// TIA Portal V19 export
FUNCTION_BLOCK "Area"   // FB100, LAD
TITLE = AREA MANAGER / ZONE CYCLE
// v1.1 : Normal Stop required added in AreaInterface
// stored: Access Published, MemoryReserve 100, SetENOAutomatically false
   VAR_INPUT
      Estop : Bool;   // Emergency stop pressed (0=OK)
      DataIn : Struct
         SelMan : Bool;   // IN: Mode selectot in AUTO position / Select Manual mode
         SelAut : Bool;   // in quale tabella di lavoro è stato copiato / Select Auto mode
         PbStart : Bool;   // IN: Push button ACKNOWLEDGE/RESET ALARMS / Pb Start Cycle
         PbStop : Bool;   // IN: Push button START CYLE / Pb Stop Cycle
         PbStopProgrammed : Bool;   // Normally not used
         PbAckRst : Bool;   // IN: Mode selectot in MANU position / Pb Reset alarms
      END_STRUCT;
      Config : "AreaConfig";
      MachinesStatus : "MachineStatus";
      ForceStopInPhase : Bool;   // Force area in stop in phase (From PLC command)
      ForceStopProgrammed : Bool;   // Force area in stop programmed (From PLC command)
      ResetTimersTimeoutStops : Bool;   // Reset timeout of stop in phase and stop programmed
   END_VAR
   VAR_OUTPUT
      AreaInterface { ExternalVisible := 'False'; ExternalWritable := 'False'} : "AreaInterface";
      DataOut : Struct
         horn : Bool;   // Area tower acustic signal
         lampReady : Bool;   // Ready for cycle lamp
         lampCycle : Bool;   // Cylce on lamp
         LampWarningPresence : Bool;   // Area tower wanring lamp
         LampAlarmPresence : Bool;   // Area tower alarm lamp
      END_STRUCT;
      SilencingAlarms : Bool;   // Command to message manager for silecing alarms
      HMI_StatusDinamicText : Int;   // Status of area for HMI
   END_VAR
   VAR
      pbStartOneShotAux : Bool;
      RstAlrOneShot1 : Bool;
      RstAlrOneShot2 : Bool;
      CycleStopImmediately : Bool;
      CycleStopInPhase : Bool;
      CycleStarted : Bool;
      CycleStopProgrammed : Bool;
      CycleOn : Bool;
      ManAuxPe : Bool;
      ManAuxNe : Bool;
      ManPositiveEdge : Bool;
      ManNegativeEdge : Bool;
      AutAuxPe : Bool;
      AutAuxNe : Bool;
      AutPositiveEdge : Bool;
      AutNegativeEdge : Bool;
      AlarmLAuxPe : Bool;
      CycleAuxPe : Bool;
      ResetAlarmsCmd : Bool;
      tonDelayPbStart { S7_SetPoint := 'True'} : IEC_TIMER;
      tonDelayRstAck { S7_SetPoint := 'True'} : IEC_TIMER;
      tonTimeOutStopPhase { S7_SetPoint := 'True'} : IEC_TIMER;
      tonTimeOutStopProgr { S7_SetPoint := 'True'} : IEC_TIMER;
      tonTimeOutResetAlr { S7_SetPoint := 'True'} : IEC_TIMER;
   END_VAR
   VAR_TEMP
      AreaEStop : Bool;
      ManMode : Bool;
      AutMode : Bool;
      pbStartOneShot : Bool;
      CycleStop : Bool;
      CycleCheckStartCnd : Bool;
      PbAckRstDelayed : Bool;
      TimeOutPT : Time;
   END_VAR
   VAR CONSTANT
      HMI_STATUS_CODE_00_INVALID : Int := 0;
      HMI_STATUS_CODE_01_EMERGENCY : Int := 1;
      HMI_STATUS_CODE_02_SEL_0 : Int := 2;
      HMI_STATUS_CODE_11_MAN : Int := 11;
      HMI_STATUS_CODE_21_AUT_NOT_READY : Int := 21;
      HMI_STATUS_CODE_22_AUT_READY : Int := 22;
      HMI_STATUS_CODE_31_CYCLE_STARTING : Int := 31;
      HMI_STATUS_CODE_32_CYCLE_ON : Int := 32;
      HMI_STATUS_CODE_41_STOP_IMMEDIATELY : Int := 41;
      HMI_STATUS_CODE_42_STOP_IN_PHASE : Int := 42;
      HMI_STATUS_CODE_43_STOP_PROGRAMMED : Int := 43;
   END_VAR
   VAR_TEMP   // added for the SCL form of the ladder/FBD networks
      _w1 : Bool;
      _w2 : Bool;
   END_VAR
BEGIN

REGION Network 1 (SCL): Info
   //=============================================================================
   //PM FORMING
   //-----------------------------------------------------------------------------
   // Library: StandardBlocks
   // Tested with: S7-1518TF
   // Engineering: TIA Portal V18
   // Restrictions: -
   // Requirements: S7-1500
   // Functionality: Area Manager
   //
   // v1.0.0  28/12/2022 
   //=============================================================================
END_REGION

REGION Network 3: EStop active
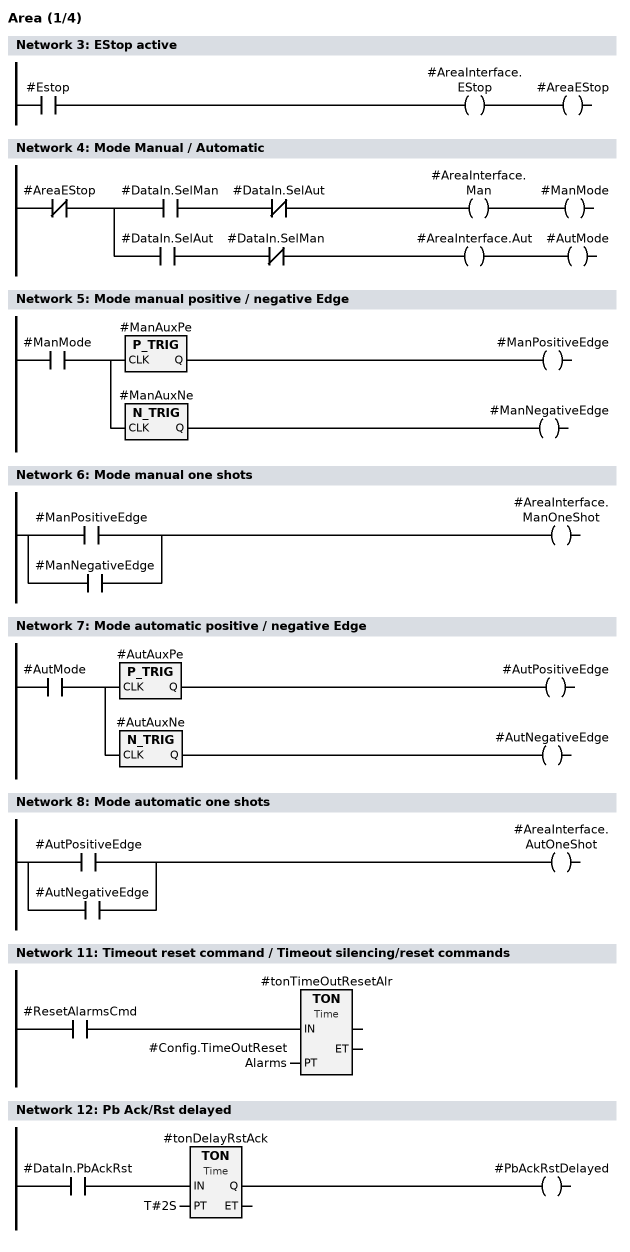
   RUNG wire#powerrail
      Contact( #Estop )
      Coil( #AreaInterface.EStop )
      Coil( #AreaEStop )
   END_RUNG
   // the same network as SCL:
   #AreaInterface.EStop := #Estop;
   #AreaEStop := #Estop;
END_REGION

REGION Network 4: Mode Manual / Automatic
   RUNG wire#powerrail
      I_Contact( #AreaEStop )
      wire#w1
      Contact( #DataIn.SelMan )
      I_Contact( #DataIn.SelAut )
      Coil( #AreaInterface.Man )
      Coil( #ManMode )
   END_RUNG
   RUNG wire#w1
      Contact( #DataIn.SelAut )
      I_Contact( #DataIn.SelMan )
      Coil( #AreaInterface.Aut )
      Coil( #AutMode )
   END_RUNG
   // the same network as SCL:
   #AreaInterface.Man := NOT #AreaEStop AND #DataIn.SelMan AND NOT #DataIn.SelAut;
   #ManMode := #AreaInterface.Man;
   #AreaInterface.Aut := NOT #AreaEStop AND #DataIn.SelAut AND NOT #DataIn.SelMan;
   #AutMode := #AreaInterface.Aut;
END_REGION

REGION Network 5: Mode manual positive / negative Edge
   RUNG wire#powerrail
      Contact( #ManMode )
      wire#w1
      P_Trig( #ManAuxPe )
      Coil( #ManPositiveEdge )
   END_RUNG
   RUNG wire#w1
      N_Trig( #ManAuxNe )
      Coil( #ManNegativeEdge )
   END_RUNG
   // the same network as SCL:
   #_w1 := #ManMode AND NOT #ManAuxPe;   // rising edge
   #ManAuxPe := #ManMode;
   #ManPositiveEdge := #_w1;
   #_w2 := NOT #ManMode AND #ManAuxNe;   // falling edge
   #ManAuxNe := #ManMode;
   #ManNegativeEdge := #_w2;
END_REGION

REGION Network 6: Mode manual one shots
   RUNG wire#powerrail
      Contact( #ManPositiveEdge )
      wire#w1
      Coil( #AreaInterface.ManOneShot )
   END_RUNG
   RUNG wire#powerrail
      Contact( #ManNegativeEdge )
   END_RUNG wire#w1
   // the same network as SCL:
   #AreaInterface.ManOneShot := #ManPositiveEdge OR #ManNegativeEdge;
END_REGION

REGION Network 7: Mode automatic positive / negative Edge
   RUNG wire#powerrail
      Contact( #AutMode )
      wire#w1
      P_Trig( #AutAuxPe )
      Coil( #AutPositiveEdge )
   END_RUNG
   RUNG wire#w1
      N_Trig( #AutAuxNe )
      Coil( #AutNegativeEdge )
   END_RUNG
   // the same network as SCL:
   #_w1 := #AutMode AND NOT #AutAuxPe;   // rising edge
   #AutAuxPe := #AutMode;
   #AutPositiveEdge := #_w1;
   #_w2 := NOT #AutMode AND #AutAuxNe;   // falling edge
   #AutAuxNe := #AutMode;
   #AutNegativeEdge := #_w2;
END_REGION

REGION Network 8: Mode automatic one shots
   RUNG wire#powerrail
      Contact( #AutPositiveEdge )
      wire#w1
      Coil( #AreaInterface.AutOneShot )
   END_RUNG
   RUNG wire#powerrail
      Contact( #AutNegativeEdge )
   END_RUNG wire#w1
   // the same network as SCL:
   #AreaInterface.AutOneShot := #AutPositiveEdge OR #AutNegativeEdge;
END_REGION

REGION Network 10: <<< ALARMS SILENCING & RESETTING >>>
END_REGION

REGION Network 11: Timeout reset command / Timeout silencing/reset commands
   RUNG wire#powerrail
      Contact( #ResetAlarmsCmd )
      { S7_Templates := "time_type := Time" } #tonTimeOutResetAlr.TON(pt := #Config.TimeOutResetAlarms, et =>)
   END_RUNG
   // the same network as SCL:
   #tonTimeOutResetAlr.TON(IN := #ResetAlarmsCmd, PT := #Config.TimeOutResetAlarms);
END_REGION

REGION Network 12: Pb Ack/Rst delayed
   RUNG wire#powerrail
      Contact( #DataIn.PbAckRst )
      { S7_Templates := "time_type := Time" } #tonDelayRstAck.TON(pt := T#2S, et =>)
      Coil( #PbAckRstDelayed )
   END_RUNG
   // the same network as SCL:
   #tonDelayRstAck.TON(IN := #DataIn.PbAckRst, PT := T#2S);
   #PbAckRstDelayed := #tonDelayRstAck.Q;
END_REGION

REGION Network 13: Alarms reset command (need ACK)
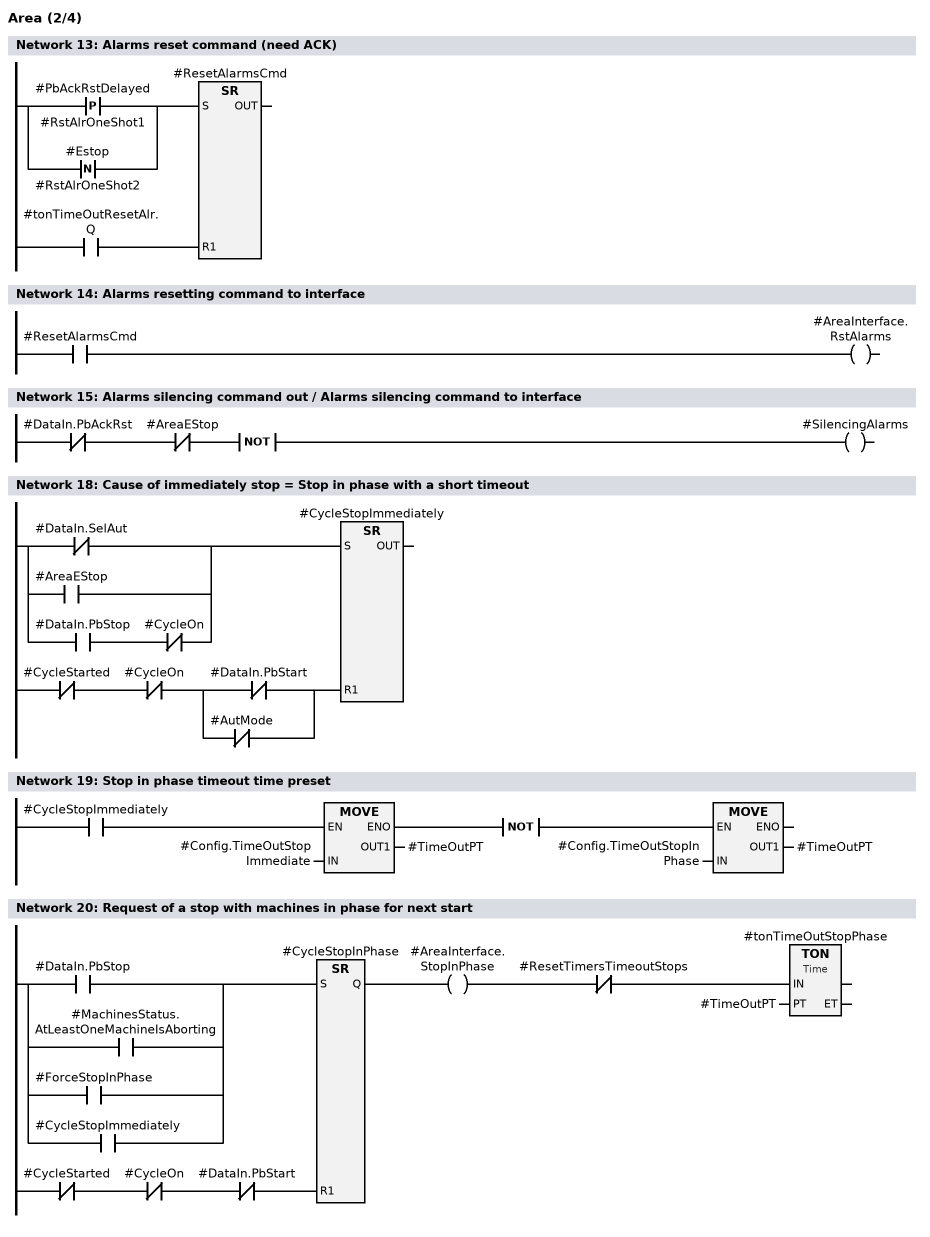
   RUNG wire#powerrail
      P_Contact(operand := #PbAckRstDelayed, bit := #RstAlrOneShot1)
      wire#w1
      S_SR(operand := #ResetAlarmsCmd, r1 := wire#w2)
   END_RUNG
   RUNG wire#powerrail
      N_Contact(operand := #Estop, bit := #RstAlrOneShot2)
   END_RUNG wire#w1
   RUNG wire#powerrail
      Contact( #tonTimeOutResetAlr.Q )
   END_RUNG wire#w2
   // the same network as SCL:
   #_w1 := #PbAckRstDelayed AND NOT #RstAlrOneShot1;   // rising edge of #PbAckRstDelayed
   #RstAlrOneShot1 := #PbAckRstDelayed;
   #_w2 := NOT #Estop AND #RstAlrOneShot2;   // falling edge of #Estop
   #RstAlrOneShot2 := #Estop;
   IF #_w1 OR #_w2 THEN
       #ResetAlarmsCmd := TRUE;   // SR flip-flop
   END_IF;
   IF #tonTimeOutResetAlr.Q THEN #ResetAlarmsCmd := FALSE; END_IF;
END_REGION

REGION Network 14: Alarms resetting command to interface
   RUNG wire#powerrail
      Contact( #ResetAlarmsCmd )
      Coil( #AreaInterface.RstAlarms )
   END_RUNG
   // the same network as SCL:
   #AreaInterface.RstAlarms := #ResetAlarmsCmd;
END_REGION

REGION Network 15: Alarms silencing command out / Alarms silencing command to interface
   RUNG wire#powerrail
      I_Contact( #DataIn.PbAckRst )
      I_Contact( #AreaEStop )
      Not()
      Coil( #SilencingAlarms )
   END_RUNG
   // the same network as SCL:
   #SilencingAlarms := NOT (NOT #DataIn.PbAckRst AND NOT #AreaEStop);
END_REGION

REGION Network 17: <<< AUTOMATIC CYCLE >>>
END_REGION

REGION Network 18: Cause of immediately stop = Stop in phase with a short timeout
   RUNG wire#powerrail
      I_Contact( #DataIn.SelAut )
      wire#w1
      S_SR(operand := #CycleStopImmediately, r1 := wire#w3)
   END_RUNG
   RUNG wire#powerrail
      Contact( #AreaEStop )
   END_RUNG wire#w1
   RUNG wire#powerrail
      Contact( #DataIn.PbStop )
      I_Contact( #CycleOn )
   END_RUNG wire#w1
   RUNG wire#powerrail
      I_Contact( #CycleStarted )
      I_Contact( #CycleOn )
      wire#w2
      I_Contact( #DataIn.PbStart )
   END_RUNG wire#w3
   RUNG wire#w2
      I_Contact( #AutMode )
   END_RUNG wire#w3
   // the same network as SCL:
   IF NOT #DataIn.SelAut OR #AreaEStop OR (#DataIn.PbStop AND NOT #CycleOn) THEN
       #CycleStopImmediately := TRUE;   // SR flip-flop
   END_IF;
   IF NOT #CycleStarted AND NOT #CycleOn AND (NOT #DataIn.PbStart OR NOT #AutMode) THEN
       #CycleStopImmediately := FALSE;
   END_IF;
END_REGION

REGION Network 19: Stop in phase timeout time preset
   RUNG wire#powerrail
      Contact( #CycleStopImmediately )
      { S7_GenerateENO := "TRUE" } Move(in := #Config.TimeOutStopImmediate, out1 => #TimeOutPT)
      Not()
      { S7_GenerateENO := "TRUE" } Move(in := #Config.TimeOutStopInPhase, out1 => #TimeOutPT)
   END_RUNG
   // the same network as SCL:
   // ENO of a box is taken as its EN; it also drops when the box reports an error
   IF #CycleStopImmediately THEN #TimeOutPT := #Config.TimeOutStopImmediate; END_IF;
   IF NOT #CycleStopImmediately THEN #TimeOutPT := #Config.TimeOutStopInPhase; END_IF;
END_REGION

REGION Network 20: Request of a stop with machines in phase for next start
   RUNG wire#powerrail
      Contact( #DataIn.PbStop )
      wire#w1
      S_SR(operand := #CycleStopInPhase, r1 := wire#w2)
      Coil( #AreaInterface.StopInPhase )
      I_Contact( #ResetTimersTimeoutStops )
      { S7_Templates := "time_type := Time" } #tonTimeOutStopPhase.TON(pt := #TimeOutPT, et =>)
   END_RUNG
   RUNG wire#powerrail
      Contact( #MachinesStatus.AtLeastOneMachineIsAborting )
   END_RUNG wire#w1
   RUNG wire#powerrail
      Contact( #ForceStopInPhase )
   END_RUNG wire#w1
   RUNG wire#powerrail
      Contact( #CycleStopImmediately )
   END_RUNG wire#w1
   RUNG wire#powerrail
      I_Contact( #CycleStarted )
      I_Contact( #CycleOn )
      I_Contact( #DataIn.PbStart )
   END_RUNG wire#w2
   // the same network as SCL:
   IF #DataIn.PbStop OR #MachinesStatus.AtLeastOneMachineIsAborting OR #ForceStopInPhase OR #CycleStopImmediately THEN
       #CycleStopInPhase := TRUE;   // SR flip-flop
   END_IF;
   IF NOT #CycleStarted AND NOT #CycleOn AND NOT #DataIn.PbStart THEN #CycleStopInPhase := FALSE; END_IF;
   #AreaInterface.StopInPhase := #CycleStopInPhase;
   #tonTimeOutStopPhase.TON(IN := #CycleStopInPhase AND NOT #ResetTimersTimeoutStops, PT := #TimeOutPT);
END_REGION

REGION Network 21: Request of a programmed stop (e.g. at the end of part)
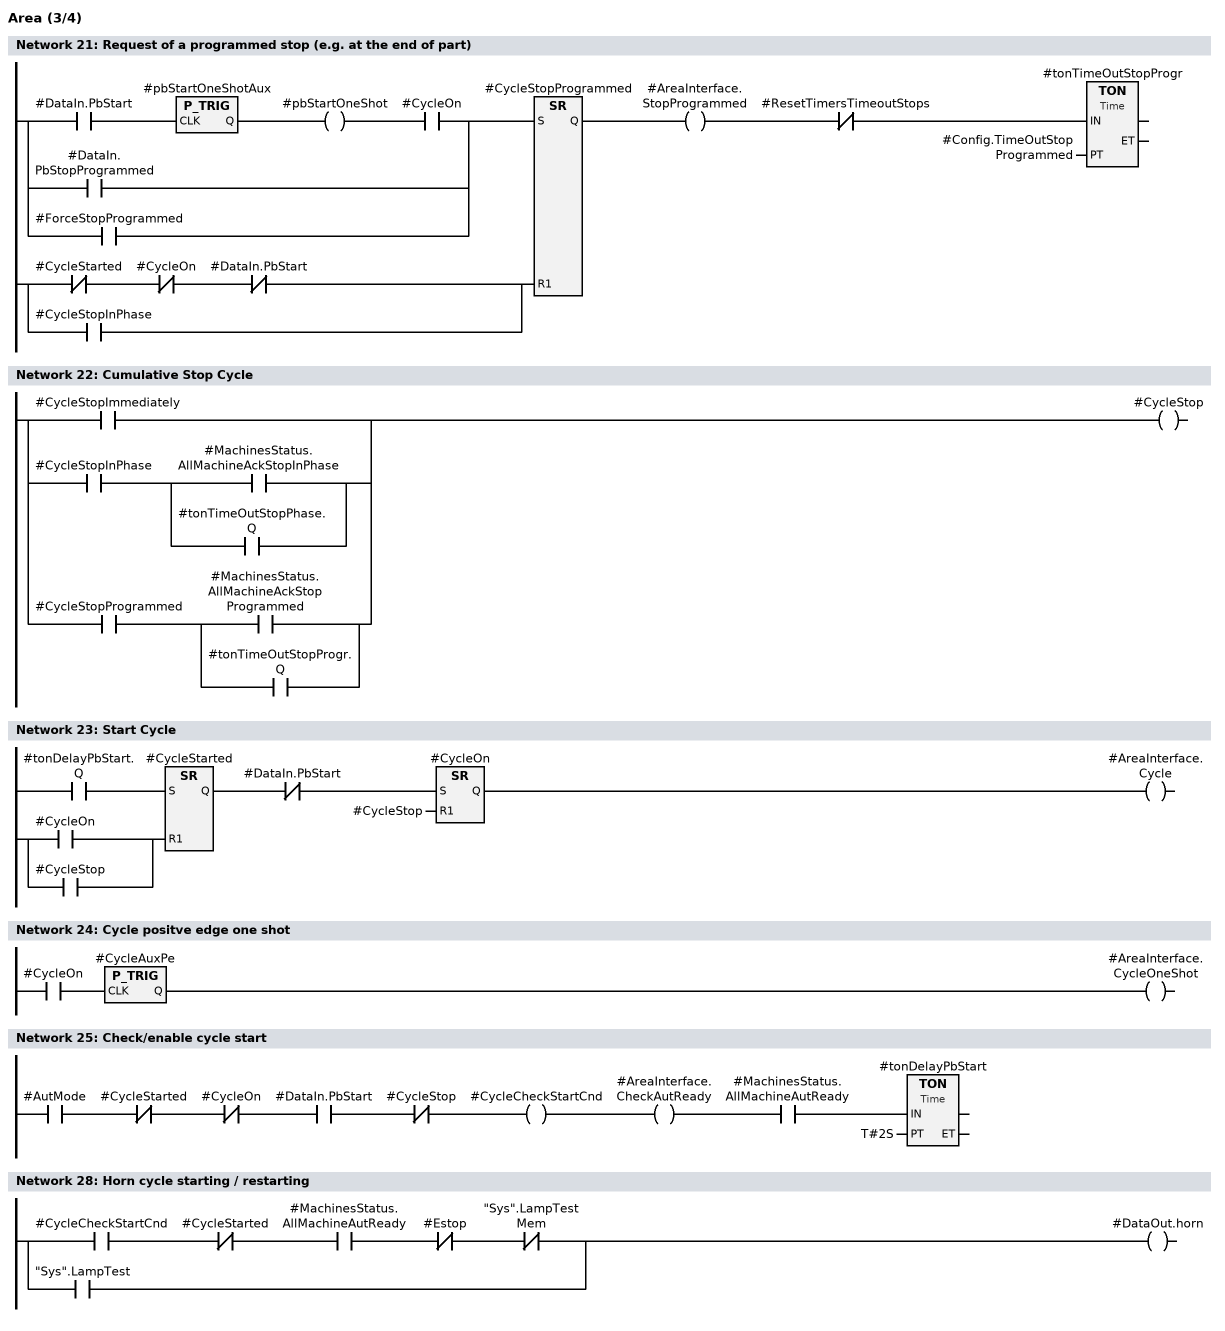
   RUNG wire#powerrail
      Contact( #DataIn.PbStart )
      P_Trig( #pbStartOneShotAux )
      Coil( #pbStartOneShot )
      Contact( #CycleOn )
      wire#w1
      S_SR(operand := #CycleStopProgrammed, r1 := wire#w2)
      Coil( #AreaInterface.StopProgrammed )
      I_Contact( #ResetTimersTimeoutStops )
      { S7_Templates := "time_type := Time" } #tonTimeOutStopProgr.TON(pt := #Config.TimeOutStopProgrammed, et =>)
   END_RUNG
   RUNG wire#powerrail
      Contact( #DataIn.PbStopProgrammed )
   END_RUNG wire#w1
   RUNG wire#powerrail
      Contact( #ForceStopProgrammed )
   END_RUNG wire#w1
   RUNG wire#powerrail
      I_Contact( #CycleStarted )
      I_Contact( #CycleOn )
      I_Contact( #DataIn.PbStart )
   END_RUNG wire#w2
   RUNG wire#powerrail
      Contact( #CycleStopInPhase )
   END_RUNG wire#w2
   // the same network as SCL:
   #_w1 := #DataIn.PbStart AND NOT #pbStartOneShotAux;   // rising edge
   #pbStartOneShotAux := #DataIn.PbStart;
   #pbStartOneShot := #_w1;
   IF (#_w1 AND #CycleOn) OR #DataIn.PbStopProgrammed OR #ForceStopProgrammed THEN
       #CycleStopProgrammed := TRUE;   // SR flip-flop
   END_IF;
   IF (NOT #CycleStarted AND NOT #CycleOn AND NOT #DataIn.PbStart) OR #CycleStopInPhase THEN
       #CycleStopProgrammed := FALSE;
   END_IF;
   #AreaInterface.StopProgrammed := #CycleStopProgrammed;
   #tonTimeOutStopProgr.TON(IN := #CycleStopProgrammed AND NOT #ResetTimersTimeoutStops,
                           PT := #Config.TimeOutStopProgrammed);
END_REGION

REGION Network 22: Cumulative Stop Cycle
   RUNG wire#powerrail
      Contact( #CycleStopImmediately )
      wire#w1
      Coil( #CycleStop )
   END_RUNG
   RUNG wire#powerrail
      Contact( #CycleStopInPhase )
      wire#w2
      Contact( #MachinesStatus.AllMachineAckStopInPhase )
   END_RUNG wire#w1
   RUNG wire#w2
      Contact( #tonTimeOutStopPhase.Q )
   END_RUNG wire#w1
   RUNG wire#powerrail
      Contact( #CycleStopProgrammed )
      wire#w3
      Contact( #MachinesStatus.AllMachineAckStopProgrammed )
   END_RUNG wire#w1
   RUNG wire#w3
      Contact( #tonTimeOutStopProgr.Q )
   END_RUNG wire#w1
   // the same network as SCL:
   #CycleStop := #CycleStopImmediately OR (#CycleStopInPhase AND (#MachinesStatus.AllMachineAckStopInPhase OR #tonTimeOutStopPhase.Q)) OR (#CycleStopProgrammed AND (#MachinesStatus.AllMachineAckStopProgrammed OR #tonTimeOutStopProgr.Q));
END_REGION

REGION Network 23: Start Cycle
   RUNG wire#powerrail
      Contact( #tonDelayPbStart.Q )
      S_SR(operand := #CycleStarted, r1 := wire#w1)
      I_Contact( #DataIn.PbStart )
      S_SR(operand := #CycleOn, r1 := #CycleStop)
      Coil( #AreaInterface.Cycle )
   END_RUNG
   RUNG wire#powerrail
      Contact( #CycleOn )
   END_RUNG wire#w1
   RUNG wire#powerrail
      Contact( #CycleStop )
   END_RUNG wire#w1
   // the same network as SCL:
   IF #tonDelayPbStart.Q THEN
       #CycleStarted := TRUE;   // SR flip-flop
   END_IF;
   IF #CycleOn OR #CycleStop THEN #CycleStarted := FALSE; END_IF;
   IF #CycleStarted AND NOT #DataIn.PbStart THEN
       #CycleOn := TRUE;   // SR flip-flop
   END_IF;
   IF #CycleStop THEN #CycleOn := FALSE; END_IF;
   #AreaInterface.Cycle := #CycleOn;
END_REGION

REGION Network 24: Cycle positve edge one shot
   RUNG wire#powerrail
      Contact( #CycleOn )
      P_Trig( #CycleAuxPe )
      Coil( #AreaInterface.CycleOneShot )
   END_RUNG
   // the same network as SCL:
   #_w1 := #CycleOn AND NOT #CycleAuxPe;   // rising edge
   #CycleAuxPe := #CycleOn;
   #AreaInterface.CycleOneShot := #_w1;
END_REGION

REGION Network 25: Check/enable cycle start
   RUNG wire#powerrail
      Contact( #AutMode )
      I_Contact( #CycleStarted )
      I_Contact( #CycleOn )
      Contact( #DataIn.PbStart )
      I_Contact( #CycleStop )
      Coil( #CycleCheckStartCnd )
      Coil( #AreaInterface.CheckAutReady )
      Contact( #MachinesStatus.AllMachineAutReady )
      { S7_Templates := "time_type := Time" } #tonDelayPbStart.TON(pt := T#2S, et =>)
   END_RUNG
   // the same network as SCL:
   #CycleCheckStartCnd := #AutMode AND NOT #CycleStarted AND NOT #CycleOn AND #DataIn.PbStart AND NOT #CycleStop;
   #AreaInterface.CheckAutReady := #CycleCheckStartCnd;
   #tonDelayPbStart.TON(IN := #CycleCheckStartCnd AND #MachinesStatus.AllMachineAutReady, PT := T#2S);
END_REGION

REGION Network 27: < OUTPUT >
   // +
   // +
   // +
   // +
   // +
   // +
   // +
   // +
   // +
   // +
END_REGION

REGION Network 28: Horn cycle starting / restarting
   RUNG wire#powerrail
      Contact( #CycleCheckStartCnd )
      I_Contact( #CycleStarted )
      Contact( #MachinesStatus.AllMachineAutReady )
      I_Contact( #Estop )
      I_Contact( "Sys".LampTestMem )
      wire#w1
      Coil( #DataOut.horn )
   END_RUNG
   RUNG wire#powerrail
      Contact( "Sys".LampTest )
   END_RUNG wire#w1
   // the same network as SCL:
   #DataOut.horn := (#CycleCheckStartCnd AND NOT #CycleStarted AND #MachinesStatus.AllMachineAutReady AND NOT #Estop AND NOT "Sys".LampTestMem) OR "Sys".LampTest;
END_REGION

REGION Network 29: Lamp automatic ready
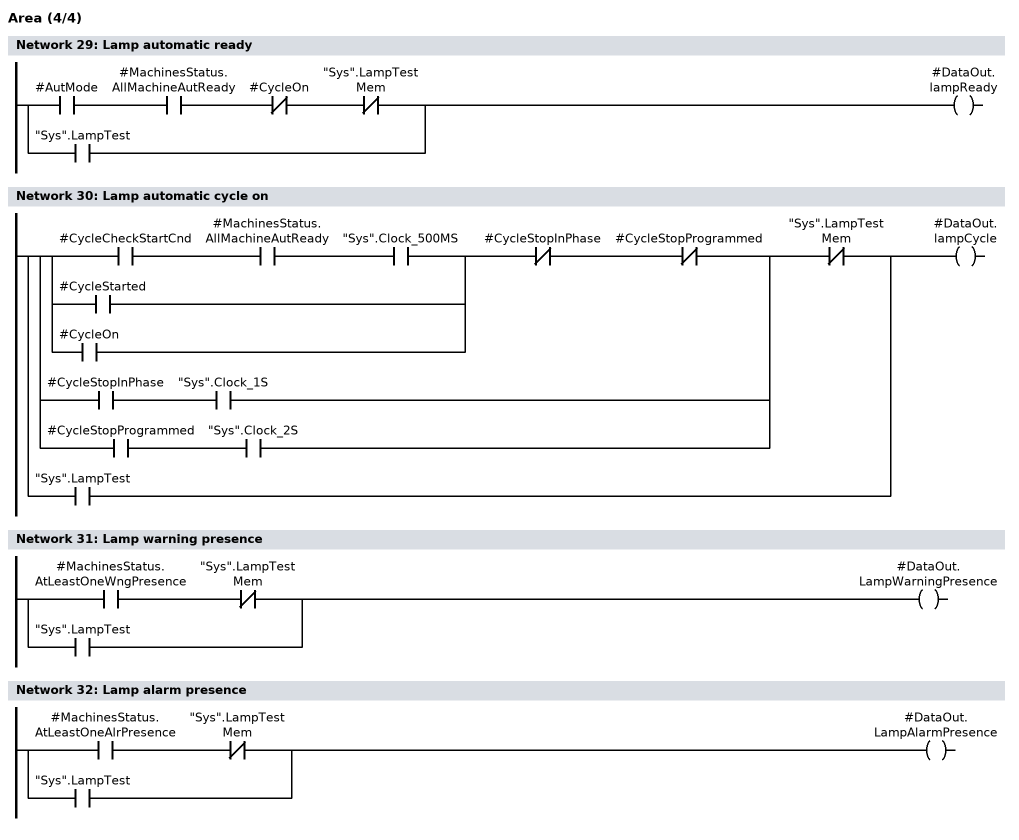
   RUNG wire#powerrail
      Contact( #AutMode )
      Contact( #MachinesStatus.AllMachineAutReady )
      I_Contact( #CycleOn )
      I_Contact( "Sys".LampTestMem )
      wire#w1
      Coil( #DataOut.lampReady )
   END_RUNG
   RUNG wire#powerrail
      Contact( "Sys".LampTest )
   END_RUNG wire#w1
   // the same network as SCL:
   #DataOut.lampReady := (#AutMode AND #MachinesStatus.AllMachineAutReady AND NOT #CycleOn AND NOT "Sys".LampTestMem) OR "Sys".LampTest;
END_REGION

REGION Network 30: Lamp automatic cycle on
   RUNG wire#powerrail
      Contact( #CycleCheckStartCnd )
      Contact( #MachinesStatus.AllMachineAutReady )
      Contact( "Sys".Clock_500MS )
      wire#w1
      I_Contact( #CycleStopInPhase )
      I_Contact( #CycleStopProgrammed )
      wire#w2
      I_Contact( "Sys".LampTestMem )
      wire#w3
      Coil( #DataOut.lampCycle )
   END_RUNG
   RUNG wire#powerrail
      Contact( #CycleStarted )
   END_RUNG wire#w1
   RUNG wire#powerrail
      Contact( #CycleOn )
   END_RUNG wire#w1
   RUNG wire#powerrail
      Contact( #CycleStopInPhase )
      Contact( "Sys".Clock_1S )
   END_RUNG wire#w2
   RUNG wire#powerrail
      Contact( #CycleStopProgrammed )
      Contact( "Sys".Clock_2S )
   END_RUNG wire#w2
   RUNG wire#powerrail
      Contact( "Sys".LampTest )
   END_RUNG wire#w3
   // the same network as SCL:
   #DataOut.lampCycle := (((((#CycleCheckStartCnd AND #MachinesStatus.AllMachineAutReady AND "Sys".Clock_500MS) OR #CycleStarted OR #CycleOn) AND NOT #CycleStopInPhase AND NOT #CycleStopProgrammed) OR (#CycleStopInPhase AND "Sys".Clock_1S) OR (#CycleStopProgrammed AND "Sys".Clock_2S)) AND NOT "Sys".LampTestMem) OR "Sys".LampTest;
END_REGION

REGION Network 31: Lamp warning presence
   RUNG wire#powerrail
      Contact( #MachinesStatus.AtLeastOneWngPresence )
      I_Contact( "Sys".LampTestMem )
      wire#w1
      Coil( #DataOut.LampWarningPresence )
   END_RUNG
   RUNG wire#powerrail
      Contact( "Sys".LampTest )
   END_RUNG wire#w1
   // the same network as SCL:
   #DataOut.LampWarningPresence := (#MachinesStatus.AtLeastOneWngPresence AND NOT "Sys".LampTestMem) OR "Sys".LampTest;
END_REGION

REGION Network 32: Lamp alarm presence
   RUNG wire#powerrail
      Contact( #MachinesStatus.AtLeastOneAlrPresence )
      I_Contact( "Sys".LampTestMem )
      wire#w1
      Coil( #DataOut.LampAlarmPresence )
   END_RUNG
   RUNG wire#powerrail
      Contact( "Sys".LampTest )
   END_RUNG wire#w1
   // the same network as SCL:
   #DataOut.LampAlarmPresence := (#MachinesStatus.AtLeastOneAlrPresence AND NOT "Sys".LampTestMem) OR "Sys".LampTest;
END_REGION

REGION Network 33 (SCL): HMI dinamic text fot Area Status
   #HMI_StatusDinamicText := #HMI_STATUS_CODE_00_INVALID;

   IF      #CycleStopImmediately THEN 
       #HMI_StatusDinamicText := #HMI_STATUS_CODE_41_STOP_IMMEDIATELY;

   ELSIF   #CycleStopInPhase THEN
       #HMI_StatusDinamicText := #HMI_STATUS_CODE_42_STOP_IN_PHASE;

   ELSIF   #CycleStopProgrammed THEN
       #HMI_StatusDinamicText := #HMI_STATUS_CODE_43_STOP_PROGRAMMED;

   ELSIF   #CycleOn THEN   
       #HMI_StatusDinamicText := #HMI_STATUS_CODE_32_CYCLE_ON;

   ELSIF  #tonDelayPbStart.IN OR #CycleStarted THEN
       #HMI_StatusDinamicText := #HMI_STATUS_CODE_31_CYCLE_STARTING;


   ELSIF   #AutMode AND #MachinesStatus.AllMachineAutReady THEN
       #HMI_StatusDinamicText := #HMI_STATUS_CODE_22_AUT_READY;

   ELSIF   #AutMode THEN
       #HMI_StatusDinamicText := #HMI_STATUS_CODE_21_AUT_NOT_READY;

   ELSIF  #Estop THEN
       #HMI_StatusDinamicText := #HMI_STATUS_CODE_01_EMERGENCY;

   ELSIF   NOT #ManMode AND NOT #AutMode THEN
       #HMI_StatusDinamicText := #HMI_STATUS_CODE_02_SEL_0;

   ELSIF   #ManMode THEN
       #HMI_StatusDinamicText := #HMI_STATUS_CODE_11_MAN;

   END_IF;
END_REGION
END_FUNCTION_BLOCK
